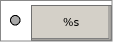
VISUALIZATION VISU_SimpleRelay  // 113x42
VAR_IN_OUT
	ref : SimpleRelay;
    widget : SimpleRelayWidget;
END_VAR
    Button (31,5 80x35), "%s", text variable: widget.text, input disabled if: ref.processes.setEnabled.statuses.enabledStatus.disabled
        OnMouseClick: execute { widget.do_request := TRUE; }
    Frame (10,10 25x30)
        shows VISU_State_gray_green(state := ref.digitalOutput)
END_VISUALIZATION

// ---- MTCS/Common/Visu/VISU_SSIEncoder.TcVIS
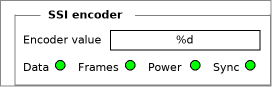
VISUALIZATION VISU_SSIEncoder  // 272x87
VAR_IN_OUT
	ref : SSIEncoder;
END_VAR
    Polyline (135,15) (270,15) (270,85) (15,85) (15,15) (40,15)
    Label (45,5 150x20), "SSI encoder"
    Rectangle (110,30 150x20), "%d", text variable: ref.counterValue
    Label (20,55 40x25), "Data"
    Frame (55,55 20x15)
        shows VISU_State_green_red(state := ref.dataError)
    Frame (125,55 20x15)
        shows VISU_State_green_red(state := ref.frameError)
    Label (75,55 50x25), "Frames"
    Label (145,55 45x25), "Power"
    Frame (190,55 20x15)
        shows VISU_State_green_red(state := ref.powerFailure)
    Frame (245,55 20x15)
        shows VISU_State_green_red(state := ref.syncError)
    Label (210,55 35x25), "Sync"
    Label (20,30 90x20), "Encoder value"
END_VISUALIZATION

// ---- MTCS/Common/Visu/VISU_State_gray_yellow.TcVIS
VISUALIZATION VISU_State_gray_yellow  // 12x17
VAR_IN_OUT
	state : BOOL;
END_VAR
    Ellipse (0,5 10x10), colour toggle: state
END_VISUALIZATION

// ---- MTCS/Common/Visu/VISU_State_gray_red.TcVIS
VISUALIZATION VISU_State_gray_red  // 12x17
VAR_IN_OUT
	state : BOOL;
END_VAR
    Ellipse (0,5 10x10), colour toggle: state
END_VISUALIZATION

// ---- MTCS/Common/Visu/VISU_State_green_gray.TcVIS
VISUALIZATION VISU_State_green_gray  // 12x17
VAR_IN_OUT
	state : BOOL;
END_VAR
    Ellipse (0,5 10x10), colour toggle: state
END_VISUALIZATION

// ---- MTCS/Common/Visu/VISU_StatusWidget.TcVIS
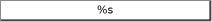
VISUALIZATION VISU_StatusWidget  // 212x22
VAR_IN_OUT
	widget : StatusWidget;
END_VAR
    Rectangle (0,0 210x20), "%s", text variable: widget.text, colour variable: widget.color.bg
        p55702900: widget.color.fg
END_VISUALIZATION

// ---- MTCS/Common/Visu/VISU_AngularAxis.TcVIS
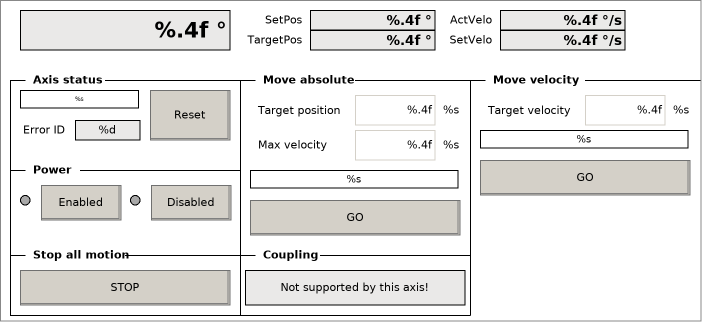
VISUALIZATION VISU_AngularAxis  // 702x322
VAR_IN_OUT
	axis : AngularAxis;
	widget : AngularAxisWidget;
END_VAR
    Rectangle (20,10 210x40), "%.4f °", text variable: axis.actPos.degrees.value
    Line (240,80) (240,315)
    Line (10,80) (10,315)
    Line (10,315) (470,315)
    Frame (10,70 230x85)
        shows VISU_BaseAxis_Status(axis := axis, axisWidget := widget.base)
    Frame (10,160 230x60)
        shows VISU_BaseAxis_Power(axis := axis, axisWidget := widget.base)
    Frame (240,70 230x170)
        shows VISU_BaseAxis_MoveAbsolute(axis := axis, axisWidget := widget.base, positionSymbol := widget.positionSymbol, velocitySymbol := widget.velocitySymbol)
    Frame (10,245 225x75)
        shows VISU_BaseAxis_Stop(axis := axis, axisWidget := widget.base)
    Line (470,80) (470,315)
    Frame (240,245 230x60)
        shows VISU_BaseAxis_Gearing(axis := axis, axisWidget := widget.base)
    Frame (470,70 230x125)
        shows VISU_BaseAxis_MoveVelocity(axis := axis, axisWidget := widget.base, positionSymbol := widget.positionSymbol, velocitySymbol := widget.velocitySymbol)
    Rectangle (310,10 125x20), "%.4f °", text variable: axis.axis_ref.NcToPlc.SetPos
    Label (255,10 50x20), "SetPos"
    Rectangle (310,30 125x20), "%.4f °", text variable: axis.axis_ref.NcToPlc.TargetPos
    Label (240,30 65x20), "TargetPos"
    Rectangle (500,10 125x20), "%.4f °/s", text variable: axis.axis_ref.NcToPlc.ActVelo
    Label (445,10 50x20), "ActVelo"
    Label (445,30 50x20), "SetVelo"
    Rectangle (500,30 125x20), "%.4f °/s", text variable: axis.axis_ref.NcToPlc.SetVelo
END_VISUALIZATION

// ---- MTCS/Common/Visu/VISU_OperatingStatus.TcVIS
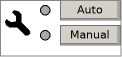
VISUALIZATION VISU_OperatingStatus  // 122x57
VAR_IN_OUT
	status : OperatingStatus;
	process : ChangeOperatingStateProcess;
END_VAR
    Frame (40,0 60x30)
        shows VISU_State_gray_green(state := status.auto)
    Button (60,0 60x20), "Auto", input disabled if: process.statuses.enabledStatus.disabled
        OnMouseClick: execute { process.set.state := OperatingStates.AUTO; process.do_request := TRUE; }
        OnMouseDown: execute {  }
    Button (60,25 60x20), "Manual", input disabled if: process.statuses.enabledStatus.disabled
        OnMouseClick: execute { process.set.state := OperatingStates.MANUAL; process.do_request := TRUE; }
        OnMouseDown: execute {  }
    Frame (40,25 36x30)
        shows VISU_State_gray_orange(state := status.manual)
    Polygon (9,27) (6,25) (5,22) (6,19) (11,22) (16,21) (16,16) (12,12) (14,10) (18,11) (21,14) (21,22) (29,30) (30,33) (28,35) (25,35) (17,27)
END_VISUALIZATION

// ---- MTCS/Common/Visu/VISU_OperatorStatus.TcVIS
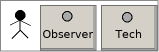
VISUALIZATION VISU_OperatorStatus  // 159x52
VAR_IN_OUT
	status : OperatorStatus;
	process : ChangeOperatorStateProcess;
END_VAR
    Line (20,30) (20,20)
    Line (12,38) (20,30)
    Line (28,38) (20,30)
    Line (20,20) (10,25)
    Line (20,20) (30,25)
    Ellipse (15,10 10x10)
    Button (101,5 56x45), "Tech", input disabled if: process.statuses.enabledStatus.disabled
        OnMouseClick: execute { process.set.state := OperatorStates.TECH; process.do_request := TRUE; }
        OnMouseDown: execute {  }
    Frame (122,7 13x20)
        shows VISU_State_gray_orange(state := status.tech)
        OnMouseClick: execute { process.set.state := OperatorStates.TECH; process.do_request := TRUE; }
    Button (40,5 56x45), "Observer", input disabled if: process.statuses.enabledStatus.disabled
        OnMouseClick: execute { process.set.state := OperatorStates.OBSERVER; process.do_request := TRUE; }
        OnMouseDown: execute {  }
    Frame (62,6 20x30)
        shows VISU_State_gray_green(state := status.observer)
        OnMouseClick: execute { process.set.state := OperatorStates.OBSERVER; process.do_request := TRUE; }
END_VISUALIZATION

// ---- MTCS/Common/Visu/VISU_OperatorStatus_Old.TcVIS
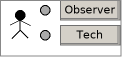
VISUALIZATION VISU_OperatorStatus_Old  // 122x57
VAR_IN_OUT
	status : OperatorStatus;
	process : ChangeOperatorStateProcess;
END_VAR
    Frame (40,0 20x30)
        shows VISU_State_gray_green(state := status.observer)
    Button (60,0 60x20), "Observer", input disabled if: process.statuses.enabledStatus.disabled
        OnMouseClick: execute { process.set.state := OperatorStates.OBSERVER; process.do_request := TRUE; }
        OnMouseDown: execute {  }
    Button (60,25 60x20), "Tech", input disabled if: process.statuses.enabledStatus.disabled
        OnMouseClick: execute { process.set.state := OperatorStates.TECH; process.do_request := TRUE; }
        OnMouseDown: execute {  }
    Frame (40,25 20x30)
        shows VISU_State_gray_orange(state := status.tech)
    Line (20,30) (20,20)
    Line (12,38) (20,30)
    Line (28,38) (20,30)
    Line (20,20) (10,25)
    Line (20,20) (30,25)
    Ellipse (15,10 10x10)
END_VISUALIZATION

// ---- MTCS/Common/Visu/VISU_State.TcVIS
VISUALIZATION VISU_State  // 12x17
VAR_IN_OUT
	state : BOOL;
	inactiveColor: Colors;
	activeColor : Colors;
END_VAR
    Ellipse (0,5 10x10), colour toggle: state, colour variable: inactiveColor
        p2167032090: activeColor
END_VISUALIZATION

// ---- MTCS/Common/Visu/VISU_State_gray_green.TcVIS
VISUALIZATION VISU_State_gray_green  // 12x17
VAR_IN_OUT
	state : BOOL;
END_VAR
    Ellipse (0,5 10x10), colour toggle: state
END_VISUALIZATION

// ---- MTCS/Common/Visu/VISU_State_gray_orange.TcVIS
VISUALIZATION VISU_State_gray_orange  // 12x17
VAR_IN_OUT
	state : BOOL;
END_VAR
    Ellipse (0,5 10x10), colour toggle: state
END_VISUALIZATION

// ---- MTCS/Common/Visu/VISU_State_green_red.TcVIS
VISUALIZATION VISU_State_green_red  // 12x17
VAR_IN_OUT
	state : BOOL;
END_VAR
    Ellipse (0,5 10x10), colour toggle: state
END_VISUALIZATION

// ---- MTCS/Common/Visu/VISU_State_red_green.TcVIS
VISUALIZATION VISU_State_red_green  // 12x17
VAR_IN_OUT
	state : BOOL;
END_VAR
    Ellipse (0,5 10x10), colour toggle: state
END_VISUALIZATION

// ---- MTCS/Common/Visu/VISU_SubSubSystemButton.TcVIS
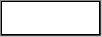
VISUALIZATION VISU_SubSubSystemButton  // 102x37
VAR_IN_OUT
    widget : SubSubSystemButtonWidget;
END_VAR
    Rectangle (0,0 100x35), invisible if: widget.isNotOrange
    Rectangle (0,0 100x35), invisible if: widget.isNotGray
    Rectangle (0,0 100x35), invisible if: widget.isNotBlue
    Rectangle (0,0 100x35), invisible if: widget.isNotRed
    Rectangle (0,0 100x35), invisible if: widget.isNotGreen
    Rectangle (0,0 100x35), "%s", text variable: widget.name
    Rectangle (0,0 100x35), invisible if: widget.notActivated
    Line (0,34) (100,34), invisible if: widget.activated
    Line (99,0) (99,35), invisible if: widget.activated
    Line (98,0) (0,0), invisible if: widget.activated
    Line (0,35) (0,0), invisible if: widget.activated
    Line (100,35) (100,1), invisible if: widget.notActivated
    Line (0,1) (99,1), invisible if: widget.notActivated
    Line (1,0) (1,35), invisible if: widget.notActivated
    Line (100,35) (1,35), invisible if: widget.notActivated
END_VISUALIZATION

// ---- MTCS/Common/Visu/VISU_SystemBackground.TcVIS
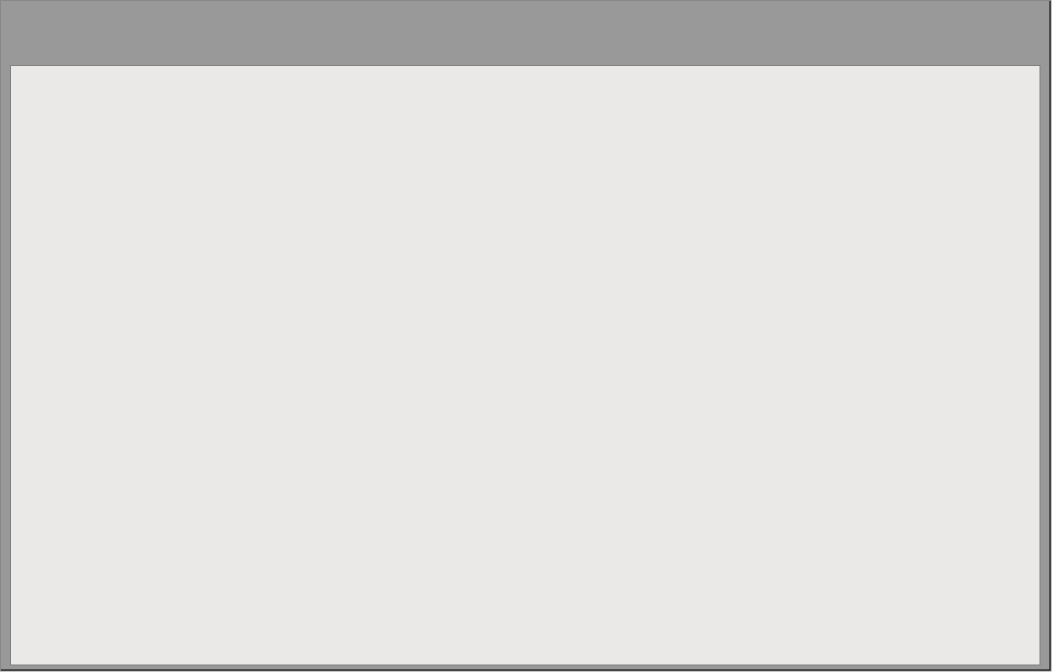
VISUALIZATION VISU_SystemBackground  // 1052x672
VAR_IN_OUT
	color : StatusColor;
END_VAR
    Rectangle (0,0 1050x670)
        p3450524324: color.bg
    Rectangle (10,65 1030x600)
END_VISUALIZATION

// ---- MTCS/Common/Visu/VISU_SystemButton.TcVIS
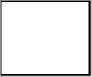
VISUALIZATION VISU_SystemButton  // 92x77
VAR_IN_OUT
    widget : SystemButtonWidget;
END_VAR
    Rectangle (0,0 90x75), invisible if: widget.isNotOrange
    Rectangle (0,0 90x75), invisible if: widget.isNotGray
    Rectangle (0,0 90x75), invisible if: widget.isNotBlue
    Rectangle (0,0 90x75), invisible if: widget.isNotRed
    Rectangle (0,0 90x75), invisible if: widget.isNotGreen
    Rectangle (0,50 90x25), "%s", text variable: widget.name
    Image (25,10 40x40), image: VISU_SystemButtonImages.Home
        p84334746: widget.name
    Rectangle (0,0 90x75), invisible if: widget.notActivated
    Line (0,74) (90,74), invisible if: widget.activated
    Line (89,75) (89,0), invisible if: widget.activated
    Line (0,74) (0,0), invisible if: widget.activated
    Line (88,0) (0,0), invisible if: widget.activated
    Line (0,1) (90,1), invisible if: widget.notActivated
    Line (1,75) (1,0), invisible if: widget.notActivated
    Line (90,75) (1,75), invisible if: widget.notActivated
    Line (90,75) (90,1), invisible if: widget.notActivated
END_VISUALIZATION

// ---- MTCS/Common/Visu/VISU_SubSystemButton.TcVIS
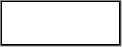
VISUALIZATION VISU_SubSystemButton  // 122x47
VAR_IN_OUT
    widget : SubSystemButtonWidget;
END_VAR
    Rectangle (0,0 120x45), invisible if: widget.isNotOrange
    Rectangle (0,0 120x45), invisible if: widget.isNotGray
    Rectangle (0,0 120x45), invisible if: widget.isNotBlue
    Rectangle (0,0 120x45), invisible if: widget.isNotRed
    Rectangle (0,0 120x45), invisible if: widget.isNotGreen
    Rectangle (0,0 120x45), "%s", text variable: widget.name
    Rectangle (0,0 120x45), invisible if: widget.notActivated
    Line (0,44) (120,44), invisible if: widget.activated
    Line (119,0) (119,45), invisible if: widget.activated
    Line (118,0) (0,0), invisible if: widget.activated
    Line (0,45) (0,0), invisible if: widget.activated
    Line (120,45) (120,1), invisible if: widget.notActivated
    Line (0,1) (119,1), invisible if: widget.notActivated
    Line (1,0) (1,45), invisible if: widget.notActivated
    Line (120,45) (1,45), invisible if: widget.notActivated
END_VISUALIZATION

// ---- MTCS/Common/Visu/VISU_SystemButton_backup.TcVIS
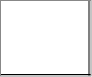
VISUALIZATION VISU_SystemButton_backup  // 92x77
VAR_IN_OUT
    widget : SystemButtonWidget;
END_VAR
    Rectangle (0,0 90x75), invisible if: widget.isNotOrange
    Rectangle (0,0 90x75), invisible if: widget.isNotGray
    Rectangle (0,0 90x75), invisible if: widget.isNotBlue
    Rectangle (0,0 90x75), invisible if: widget.isNotRed
    Rectangle (0,0 90x75), invisible if: widget.isNotGreen
    Rectangle (0,50 90x25), "%s", text variable: widget.name
    Image (25,10 40x40), image: VISU_SystemButtonImages.Home
        p84334746: widget.name
    Rectangle (0,0 90x75), invisible if: widget.notActivated
    Line (0,74) (90,74)
    Line (89,75) (89,0)
    Line (0,74) (0,0)
    Line (88,0) (0,0)
END_VISUALIZATION

// ---- MTCS/Common/Visu/VISU_SystemControl.TcVIS
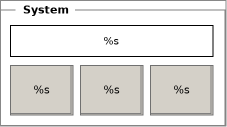
VISUALIZATION VISU_SystemControl  // 227x127
VAR_IN_OUT
    status : StatusWidget;
	button_initialize : InitializeButtonWidget;
    button_operating : OperatingButtonWidget;
    button_locking : LockingButtonWidget;
END_VAR
    Polyline (15,10) (0,10) (0,125) (225,125) (225,10) (75,10)
    Button (150,65 63x50), "%s", text variable: button_operating.text, input disabled if: button_operating.deactivate
        OnMouseClick: execute { button_operating.do_request := TRUE; }
    Button (80,65 63x50), "%s", text variable: button_locking.text, input disabled if: button_locking.deactivate
        OnMouseClick: execute { button_locking.do_request := TRUE; }
    Frame (10,25 205x35)
        shows VISU_StatusWidget(widget := status)
    Button (10,65 63x50), "%s", text variable: button_initialize.text, input disabled if: button_initialize.deactivate
        OnMouseClick: execute { button_initialize.do_request := TRUE; }
    Label (20,0 55x20), "System"
END_VISUALIZATION

// ---- MTCS/Common/Widgets/LimitSwitchesTextList.TcTLO
TEXTLIST LimitSwitchesTextList
  0 = 'Positive'
  1 = 'Negative'
   = ''
END_TEXTLIST

// ---- MTCS/Cover/Visu/VISU_Cover.TcVIS
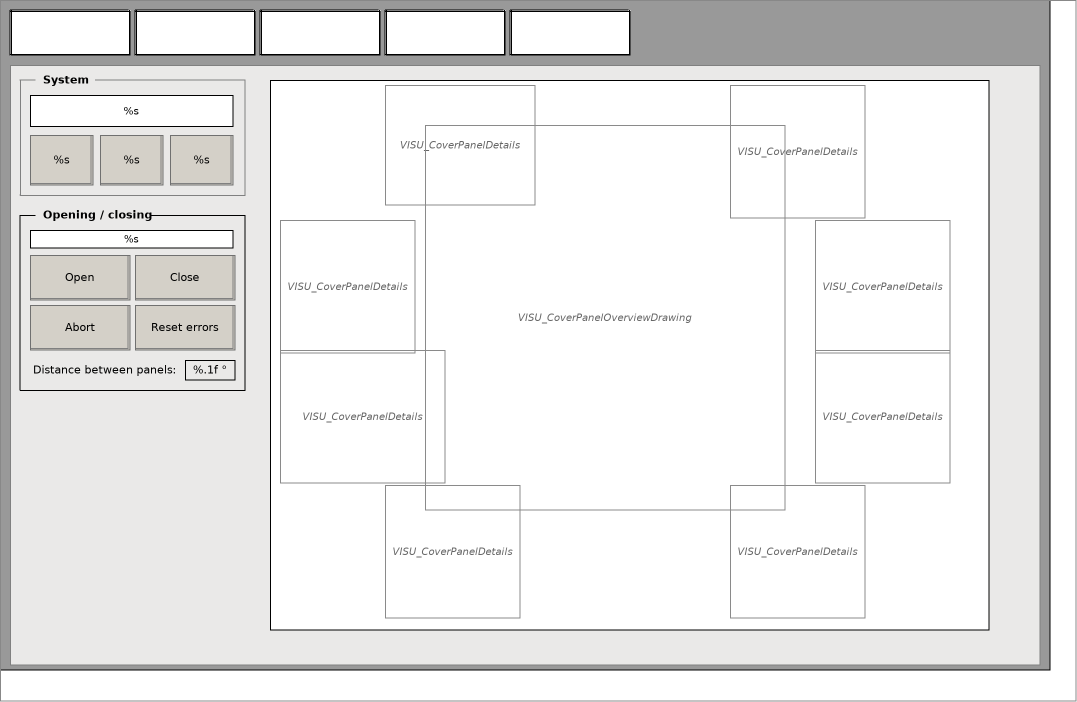
VISUALIZATION VISU_Cover  // 1077x702
VAR_IN_OUT
	ref : Cover;
    widget : CoverWidget;
END_VAR
    Frame (0,0 1075x700)
        shows VISU_SystemBackground(color := widget.actualStatus.color)
    Frame (10,65 1005x535)
        shows VISU_COVER_OVERVIEW(cover := ref, coverWidget := widget)
        shows VISU_CoverPanelSet(config := ref.config.top, set := ref.parts.top, widget := widget.top, currentMeasurement := ref.currentMeasurement)
        shows VISU_CoverPanelSet(config := ref.config.bottom, set := ref.parts.bottom, widget := widget.bottom, currentMeasurement := ref.currentMeasurement)
        shows VISU_CoverIO(io := ref.parts.io, widget := widget.io)
        shows VISU_CoverConfig(editableConfig := ref.editableConfig, activeConfig := ref.config, mgr := ref.parts.configManager, mgrWidget := widget.configManager, activeTab := widget.activeConfigTab)
    Frame (10,10 120x40)
        shows VISU_SubSystemButton(widget := widget.button_overview)
        OnMouseClick: FrameSelectionChange Selection=SelectedFrame=804c056d-b005-490b-b68c-1832c22506a3, GlobSel=AssignType=Directly, SelType=Locally
        OnMouseClick: execute { widget.activeTab := CoverTabs.OVERVIEW; }
    Frame (135,10 120x40)
        shows VISU_SubSystemButton(widget := widget.button_top)
        OnMouseClick: FrameSelectionChange Selection=SelectedFrame=804c056d-b005-490b-b68c-1832c22506a3, Selection=1, GlobSel=AssignType=Directly, SelType=Locally
        OnMouseClick: execute { widget.activeTab := CoverTabs.TOP; }
    Frame (260,10 120x40)
        shows VISU_SubSystemButton(widget := widget.button_bottom)
        OnMouseClick: FrameSelectionChange Selection=SelectedFrame=804c056d-b005-490b-b68c-1832c22506a3, Selection=2, GlobSel=AssignType=Directly, SelType=Locally
        OnMouseClick: execute { widget.activeTab := CoverTabs.BOTTOM; }
    Frame (385,10 120x40)
        shows VISU_SubSystemButton(widget := widget.button_io)
        OnMouseClick: FrameSelectionChange Selection=SelectedFrame=804c056d-b005-490b-b68c-1832c22506a3, Selection=3, GlobSel=AssignType=Directly, SelType=Locally
        OnMouseClick: execute { widget.activeTab := CoverTabs.IO; }
    Frame (510,10 120x40)
        shows VISU_SubSystemButton(widget := widget.button_config)
        OnMouseClick: FrameSelectionChange Selection=SelectedFrame=804c056d-b005-490b-b68c-1832c22506a3, Selection=4, GlobSel=AssignType=Directly, SelType=Locally
        OnMouseClick: execute { widget.activeTab := CoverTabs.CONFIG; }
END_VISUALIZATION

// ---- MTCS/Cover/Visu/VISU_CoverConfig_General.TcVIS
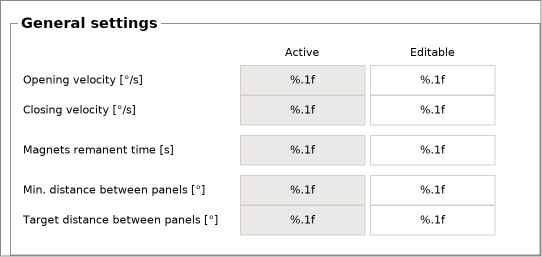
VISUALIZATION VISU_CoverConfig_General  // 542x257
VAR_IN_OUT
	activeConfig : CoverConfig;
    editableConfig : CoverConfig;
END_VAR
    GroupBox (10,15 530x240), "General settings"
        Label (10,50 175x30), "Opening velocity [°/s]"
        Label (10,80 175x30), "Closing velocity [°/s]"
        Label (10,160 190x30), "Min. distance between panels [°]"
        Label (360,25 125x25), "Editable"
        Label (230,25 125x25), "Active"
        Label (10,120 175x30), "Magnets remanent time [s]"
        Label (10,190 205x30), "Target distance between panels [°]"
        Frame (230,160 279x35)
            shows VISU_ConfigLREAL1Entry(active := activeConfig.minDistanceBetweenPanelSets, editable := editableConfig.minDistanceBetweenPanelSets)
        Frame (230,190 279x40)
            shows VISU_ConfigLREAL1Entry(active := activeConfig.targetDistanceBetweenPanelSets, editable := editableConfig.targetDistanceBetweenPanelSets)
        Frame (230,120 279x35)
            shows VISU_ConfigLREAL1Entry(active := activeConfig.magnetRemanentTime, editable := editableConfig.magnetRemanentTime)
        Frame (230,50 255x35)
            shows VISU_ConfigLREAL1Entry(active := activeConfig.openingVelocity, editable := editableConfig.openingVelocity)
        Frame (230,80 255x35)
            shows VISU_ConfigLREAL1Entry(active := activeConfig.closingVelocity, editable := editableConfig.closingVelocity)
END_VISUALIZATION

// ---- MTCS/Cover/Visu/VISU_CoverConfig.TcVIS
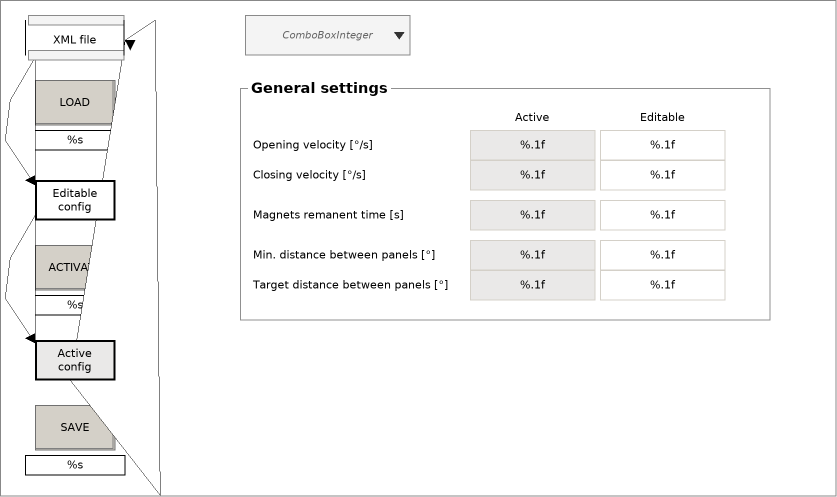
VISUALIZATION VISU_CoverConfig  // 837x497
VAR_IN_OUT
    editableConfig : CoverConfig;
	activeConfig : CoverConfig;
    mgr : ConfigManager;
    mgrWidget : ConfigManagerWidget;
    activeTab : CoverConfigTabs;
END_VAR
    Frame (10,5 190x490)
        shows VISU_ConfigManager(mgr := mgr, widget := mgrWidget)
    ComboBoxInteger (245,15 165x40), variable: activeTab, text list: 'CoverConfigTabsTextList'
    Frame (230,65 605x430), frame switch variable: activeTab
        shows VISU_CoverConfig_General(activeConfig := activeConfig, editableConfig := editableConfig)
        shows VISU_CoverConfig_PanelSet(activeConfig := activeConfig.top, editableConfig := editableConfig.top)
        shows VISU_CoverConfig_PanelSet(activeConfig := activeConfig.bottom, editableConfig := editableConfig.bottom)
        shows VISU_CoverConfig_Panel(activeConfig := activeConfig.top.p1, editableConfig := editableConfig.top.p1)
        shows VISU_CoverConfig_Panel(activeConfig := activeConfig.top.p2, editableConfig := editableConfig.top.p2)
        shows VISU_CoverConfig_Panel(activeConfig := activeConfig.top.p3, editableConfig := editableConfig.top.p3)
        shows VISU_CoverConfig_Panel(activeConfig := activeConfig.top.p4, editableConfig := editableConfig.top.p4)
        shows VISU_CoverConfig_Panel(activeConfig := activeConfig.bottom.p1, editableConfig := editableConfig.bottom.p1)
        shows VISU_CoverConfig_Panel(activeConfig := activeConfig.bottom.p2, editableConfig := editableConfig.bottom.p2)
        shows VISU_CoverConfig_Panel(activeConfig := activeConfig.bottom.p3, editableConfig := editableConfig.bottom.p3)
        shows VISU_CoverConfig_Panel(activeConfig := activeConfig.bottom.p4, editableConfig := editableConfig.bottom.p4)
END_VISUALIZATION

// ---- MTCS/Cover/Visu/VISU_CoverConfig_PanelSet.TcVIS
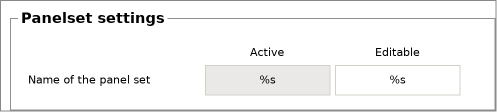
VISUALIZATION VISU_CoverConfig_PanelSet  // 497x112
VAR_IN_OUT
	activeConfig : CoverPanelSetConfig;
	editableConfig : CoverPanelSetConfig;
END_VAR
    GroupBox (10,10 485x100), "Panelset settings"
        Label (325,30 125x25), "Editable"
        Label (195,30 125x25), "Active"
        Frame (195,55 255x30)
            shows VISU_ConfigStringEntry(active := activeConfig.name, editable := editableConfig.name)
        Label (15,55 175x30), "Name of the panel set"
END_VISUALIZATION

// ---- MTCS/Cover/Visu/VISU_COVER_OVERVIEW.TcVIS
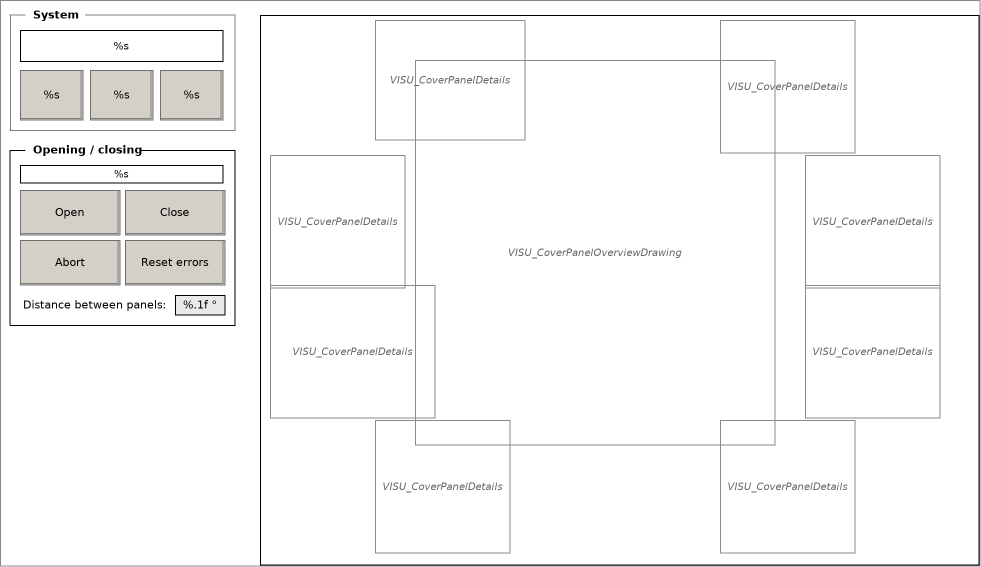
VISUALIZATION VISU_COVER_OVERVIEW  // 981x567
VAR_IN_OUT
	cover : Cover;
	coverWidget : CoverWidget;
END_VAR
    Rectangle (260,15 719x550)
    Frame (720,20 135x133)
        shows VISU_CoverPanelDetails(config := cover.config.top.p1, panel := cover.parts.top.parts.p1, widget := coverWidget.top.p1, magnetEnabled := cover.parts.top.parts.magnetsRelay.digitalOutput)
        pReferences[0]: name='Top 1'
    Frame (805,155 135x133)
        shows VISU_CoverPanelDetails(config := cover.config.bottom.p1, panel := cover.parts.bottom.parts.p1, widget := coverWidget.bottom.p1, magnetEnabled := cover.parts.bottom.parts.magnetsRelay.digitalOutput)
        pReferences[0]: name='Top 1'
    Frame (805,285 135x133)
        shows VISU_CoverPanelDetails(config := cover.config.top.p2, panel := cover.parts.top.parts.p2, widget := coverWidget.top.p2, magnetEnabled := cover.parts.top.parts.magnetsRelay.digitalOutput)
        pReferences[0]: name='Top 1'
    Frame (720,420 135x133)
        shows VISU_CoverPanelDetails(config := cover.config.bottom.p2, panel := cover.parts.bottom.parts.p2, widget := coverWidget.bottom.p2, magnetEnabled := cover.parts.bottom.parts.magnetsRelay.digitalOutput)
        pReferences[0]: name='Top 1'
    Frame (375,20 150x120)
        shows VISU_CoverPanelDetails(config := cover.config.bottom.p4, panel := cover.parts.bottom.parts.p4, widget := coverWidget.bottom.p4, magnetEnabled := cover.parts.bottom.parts.magnetsRelay.digitalOutput)
        pReferences[0]: name='Top 1'
    Frame (270,155 135x133)
        shows VISU_CoverPanelDetails(config := cover.config.top.p4, panel := cover.parts.top.parts.p4, widget := coverWidget.top.p4, magnetEnabled := cover.parts.top.parts.magnetsRelay.digitalOutput)
        pReferences[0]: name='Top 1'
    Frame (270,285 165x133)
        shows VISU_CoverPanelDetails(config := cover.config.bottom.p3, panel := cover.parts.bottom.parts.p3, widget := coverWidget.bottom.p3, magnetEnabled := cover.parts.bottom.parts.magnetsRelay.digitalOutput)
        pReferences[0]: name='Top 1'
    Frame (375,420 135x133)
        shows VISU_CoverPanelDetails(config := cover.config.top.p3, panel := cover.parts.top.parts.p3, widget := coverWidget.top.p3, magnetEnabled := cover.parts.top.parts.magnetsRelay.digitalOutput)
        pReferences[0]: name='Top 1'
    Frame (415,60 360x385)
        shows VISU_CoverPanelOverviewDrawing(cover := cover, coverWidget := coverWidget)
    Frame (10,5 208x95)
        shows VISU_SystemControl(status := coverWidget.actualStatus, button_initialize := coverWidget.button_initialize, button_operating := coverWidget.button_operating, button_locking := coverWidget.button_locking)
    Frame (20,165 205x20)
        shows VISU_StatusWidget(widget := coverWidget.apertureProcedureStatus)
    Button (20,190 100x45), "Open", input disabled if: cover.processes.open.statuses.enabledStatus.disabled
        OnMouseClick: execute { cover.processes.open.do_request := TRUE; }
    Button (125,190 100x45), "Close", input disabled if: cover.processes.close.statuses.enabledStatus.disabled
        OnMouseClick: execute { cover.processes.close.do_request := TRUE; }
    Button (20,240 100x45), "Abort", input disabled if: cover.processes.abort.statuses.enabledStatus.disabled
        OnMouseClick: execute { cover.processes.abort.do_request := TRUE; }
    Button (125,240 100x45), "Reset errors", input disabled if: cover.processes.reset.statuses.enabledStatus.disabled
        OnMouseClick: execute { cover.processes.reset.do_request := TRUE; }
    Rectangle (175,295 50x20), "%.1f °", text variable: cover.parts.apertureProcedure.distance.degrees.value
    Label (20,290 150x30), "Distance between panels:"
    Line (10,150) (25,150)
    Label (30,140 105x20), "Opening / closing"
    Line (140,150) (235,150)
    Line (235,325) (235,150)
    Line (10,325) (10,150)
    Line (10,325) (235,325)
END_VISUALIZATION

// ---- MTCS/Cover/Widgets/CoverConfigTabsTextList.TcTLO
TEXTLIST CoverConfigTabsTextList
  0 = 'General'
  1 = 'Top'
  2 = 'Bottom'
  3 = 'Top panel 1'
  4 = 'Top panel 2'
  5 = 'Top panel 3'
  6 = 'Top panel 4'
  7 = 'Bottom panel 1'
  8 = 'Bottom panel 2'
  9 = 'Bottom panel 3'
  10 = 'Bottom panel 4'
   = ''
END_TEXTLIST

// ---- MTCS/Hydraulics/Widgets/HydraulicsConfigTabsTextList.TcTLO
TEXTLIST HydraulicsConfigTabsTextList
  0 = 'General'
  1 = 'Top side - general'
  2 = 'Top side - pressure measurement'
  3 = 'Top side - frequency measurement'
  4 = 'Bottom side - general'
  5 = 'Bottom side - pressure measurement'
  6 = 'Bottom side - frequency measurement'
   = ''
END_TEXTLIST

// ---- MTCS/M1/Widgets/M1ConfigTabsTextList.TcTLO
TEXTLIST M1ConfigTabsTextList
  0 = 'General'
  1 = 'Radial - General'
  2 = 'Radial - Pressure @ regulator'
  3 = 'Radial - Pressure @ mirror cell'
  4 = 'Axial - General'
  5 = 'Axial - Pressure @ regulator'
  6 = 'Axial - Pressure @ mirror cell'
  7 = 'Axial - Force sensors'
  8 = 'Axial - Average force'
  9 = 'Inclinometer - voltage'
   = ''
END_TEXTLIST

// ---- VISUs/VISU_MAIN.TcVIS
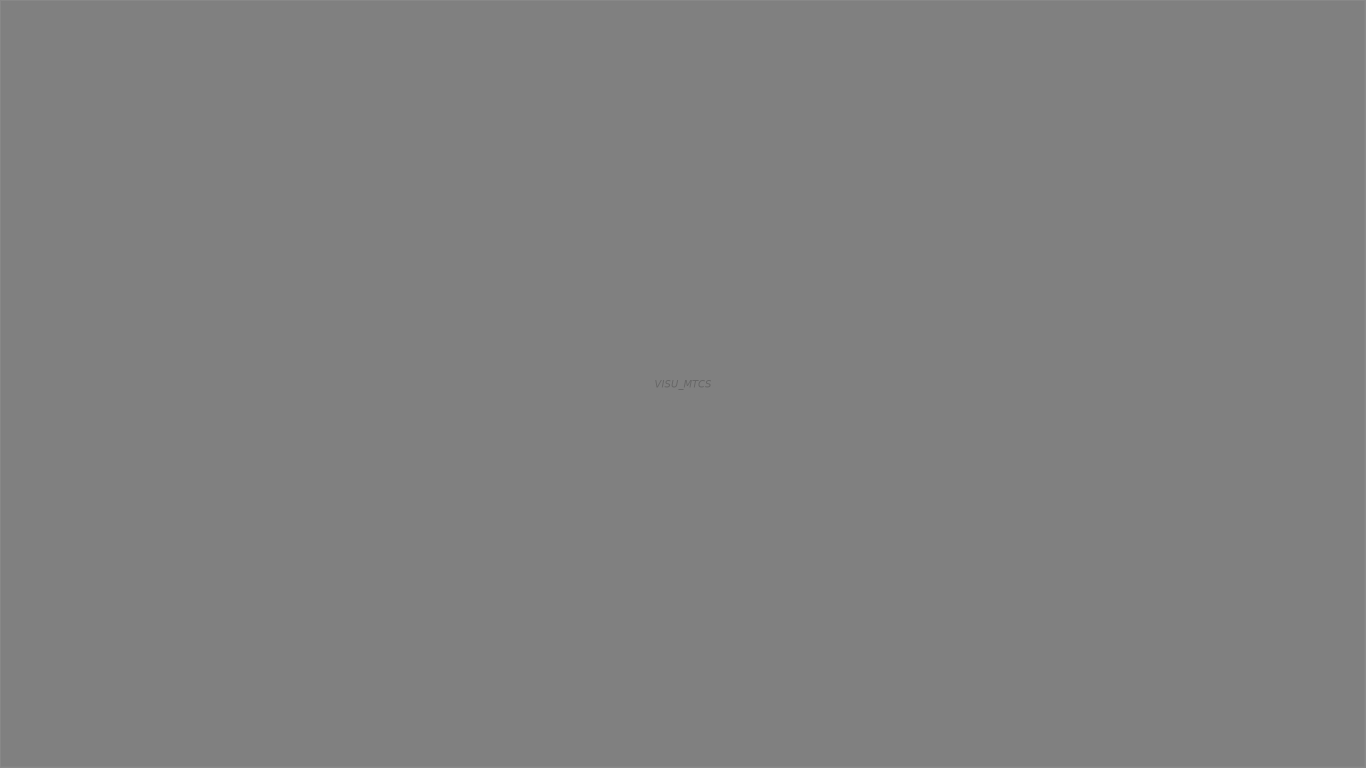
VISUALIZATION VISU_MAIN  // 1366x768
    Frame (0,0 1366x768)
        shows VISU_MTCS(mtcs := GLOBAL.mtcs, mtcsWidget := GLOBAL.gui)
        shows VISU_MTCSBlankScreen(widget := GLOBAL.gui.blankScreen)
END_VISUALIZATION
